// TIA Portal V20 export
FUNCTION "03 T4 LANT Aux" : Void   // FC1312, LAD
TITLE = AUXILIARIES
{ S7_Optimized_Access := 'TRUE' }
// stored: AutoNumber false, SetENOAutomatically false
   VAR_TEMP
      Aux_OS : Bool;
      Aux_sup : Real;
      Aux_inf : Real;
      Aux_DInt : DInt;
      Aux_Real : Real;
   END_VAR
   VAR CONSTANT
      "Max differenza L tubi" : Real := 500.0;
   END_VAR
   VAR_TEMP   // added for the SCL form of the ladder/FBD networks
      _w1 : Bool;
      _w2 : Bool;
   END_VAR
BEGIN

REGION Network 1: =========== MEMORIES ===========
END_REGION

REGION Network 2: TimeOutBancal: Calcul TimeOut
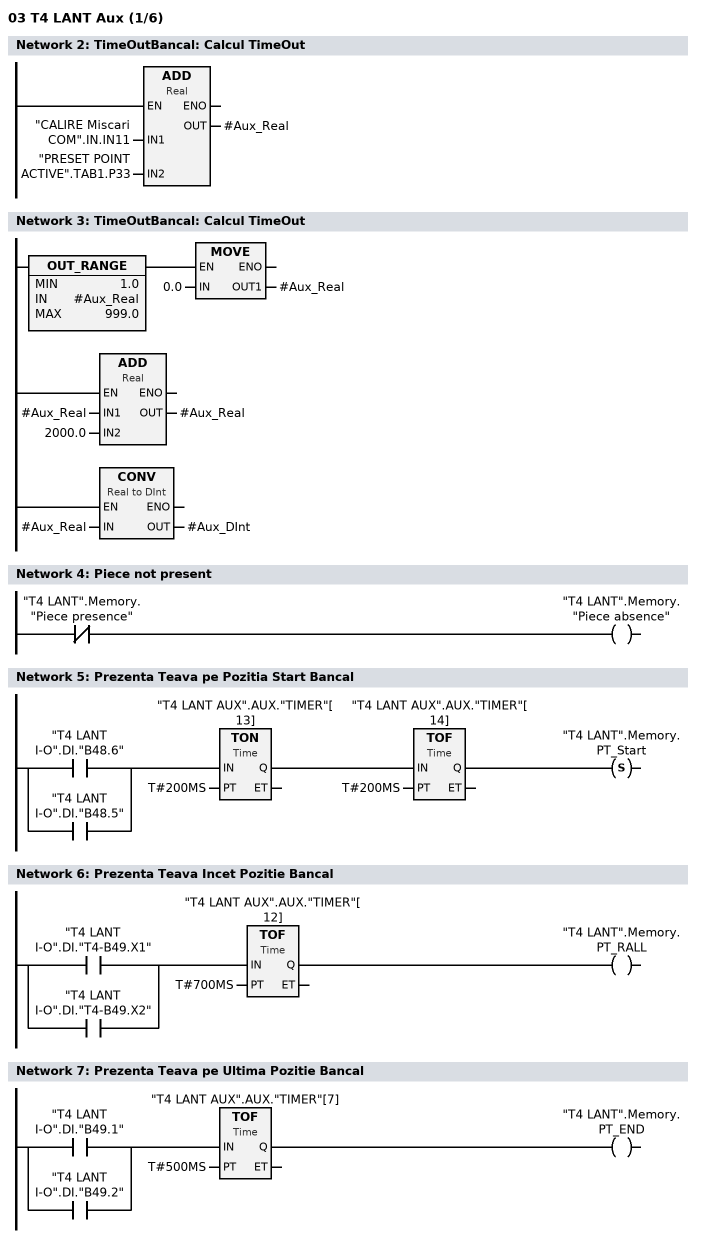
   RUNG wire#powerrail
      { S7_Templates := "SrcType := Real" } Add(in1 := "CALIRE Miscari COM".IN.IN11, in2 := "PRESET POINT ACTIVE".TAB1.P33, out => #Aux_Real)
   END_RUNG
   // the same network as SCL:
   #Aux_Real := "CALIRE Miscari COM".IN.IN11 + "PRESET POINT ACTIVE".TAB1.P33;
END_REGION

REGION Network 3: TimeOutBancal: Calcul TimeOut
   IF (#Aux_Real < 1.0) OR (#Aux_Real > 999.0) THEN #Aux_Real := 0.0; END_IF;
   #Aux_Real := #Aux_Real + 2000.0;
   #Aux_DInt := REAL_TO_DINT(#Aux_Real);
END_REGION

REGION Network 4: Piece not present
   RUNG wire#powerrail
      I_Contact( "T4 LANT".Memory."Piece presence" )
      Coil( "T4 LANT".Memory."Piece absence" )
   END_RUNG
   // the same network as SCL:
   "T4 LANT".Memory."Piece absence" := NOT "T4 LANT".Memory."Piece presence";
END_REGION

REGION Network 5: Prezenta Teava pe Pozitia Start Bancal
   RUNG wire#powerrail
      Contact( "T4 LANT I-O".DI."B48.6" )
      wire#w1
      { S7_Templates := "time_type := Time" } "T4 LANT AUX".AUX."TIMER"[13].TON(pt := T#200MS, et =>)
      { S7_Templates := "time_type := Time" } "T4 LANT AUX".AUX."TIMER"[14].TOF(pt := T#200MS, et =>)
      S_Coil( "T4 LANT".Memory.PT_Start )
   END_RUNG
   RUNG wire#powerrail
      Contact( "T4 LANT I-O".DI."B48.5" )
   END_RUNG wire#w1
   // the same network as SCL:
   "T4 LANT AUX".AUX."TIMER"[13].TON(IN := "T4 LANT I-O".DI."B48.6" OR "T4 LANT I-O".DI."B48.5", PT := T#200MS);
   "T4 LANT AUX".AUX."TIMER"[14].TOF(IN := "T4 LANT AUX".AUX."TIMER"[13].Q, PT := T#200MS);
   IF "T4 LANT AUX".AUX."TIMER"[14].Q THEN "T4 LANT".Memory.PT_Start := TRUE; END_IF;
END_REGION

REGION Network 6: Prezenta Teava Incet Pozitie Bancal
   RUNG wire#powerrail
      Contact( "T4 LANT I-O".DI."T4-B49.X1" )
      wire#w1
      { S7_Templates := "time_type := Time" } "T4 LANT AUX".AUX."TIMER"[12].TOF(pt := T#700MS, et =>)
      Coil( "T4 LANT".Memory.PT_RALL )
   END_RUNG
   RUNG wire#powerrail
      Contact( "T4 LANT I-O".DI."T4-B49.X2" )
   END_RUNG wire#w1
   // the same network as SCL:
   "T4 LANT AUX".AUX."TIMER"[12].TOF(IN := "T4 LANT I-O".DI."T4-B49.X1" OR "T4 LANT I-O".DI."T4-B49.X2",
                           PT := T#700MS);
   "T4 LANT".Memory.PT_RALL := "T4 LANT AUX".AUX."TIMER"[12].Q;
END_REGION

REGION Network 7: Prezenta Teava pe Ultima Pozitie Bancal
   RUNG wire#powerrail
      Contact( "T4 LANT I-O".DI."B49.1" )
      wire#w1
      { S7_Templates := "time_type := Time" } "T4 LANT AUX".AUX."TIMER"[7].TOF(pt := T#500MS, et =>)
      Coil( "T4 LANT".Memory.PT_END )
   END_RUNG
   RUNG wire#powerrail
      Contact( "T4 LANT I-O".DI."B49.2" )
   END_RUNG wire#w1
   // the same network as SCL:
   "T4 LANT AUX".AUX."TIMER"[7].TOF(IN := "T4 LANT I-O".DI."B49.1" OR "T4 LANT I-O".DI."B49.2", PT := T#500MS);
   "T4 LANT".Memory.PT_END := "T4 LANT AUX".AUX."TIMER"[7].Q;
END_REGION

REGION Network 8: T4-Lant: LAnt in Pozitia 'Pas'
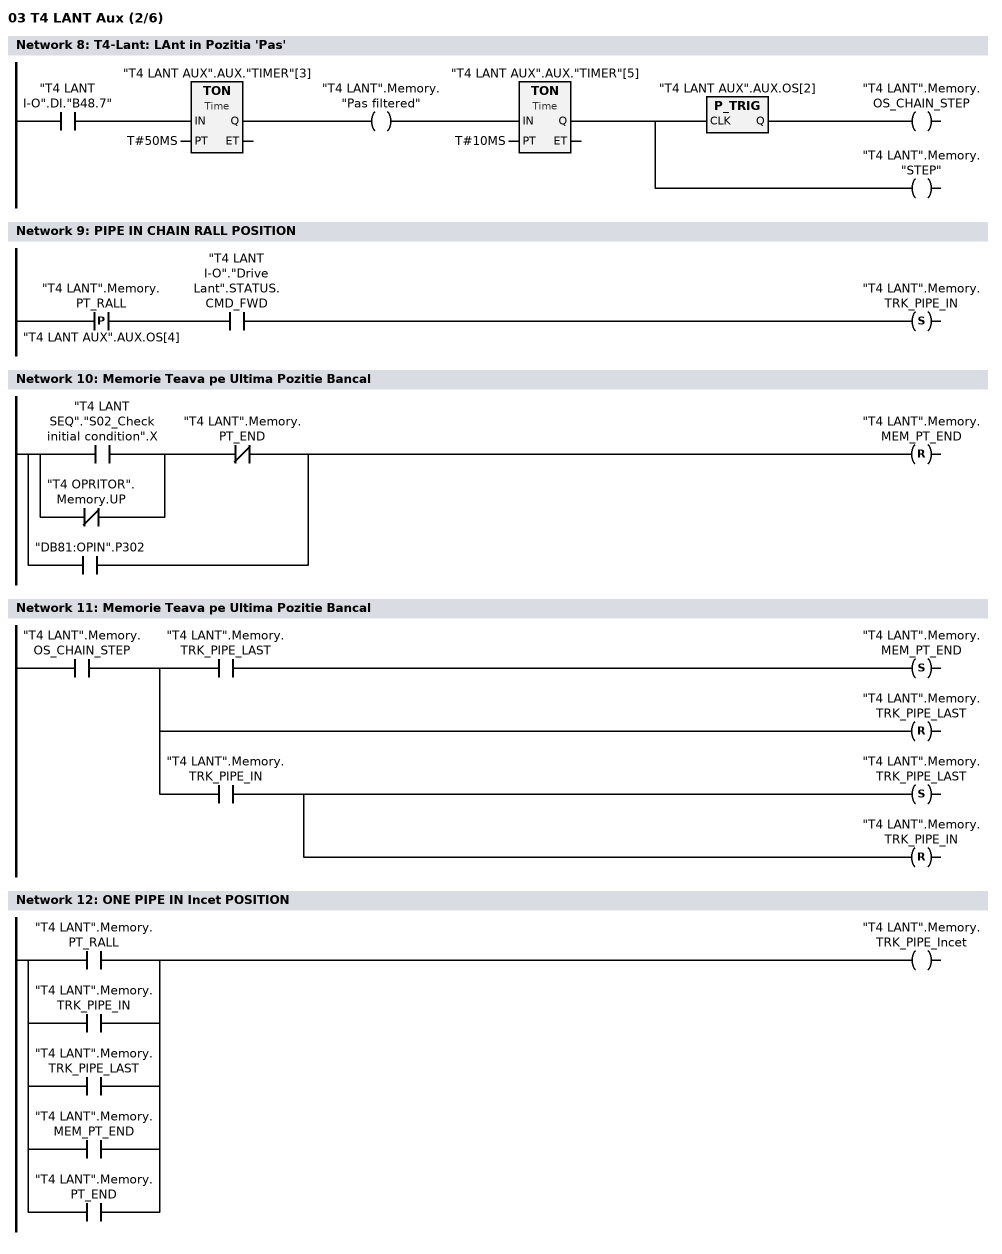
   RUNG wire#powerrail
      Contact( "T4 LANT I-O".DI."B48.7" )
      { S7_Templates := "time_type := Time" } "T4 LANT AUX".AUX."TIMER"[3].TON(pt := T#50MS, et =>)
      Coil( "T4 LANT".Memory."Pas filtered" )
      { S7_Templates := "time_type := Time" } "T4 LANT AUX".AUX."TIMER"[5].TON(pt := T#10MS, et =>)
      wire#w1
      P_Trig( "T4 LANT AUX".AUX.OS[2] )
      Coil( "T4 LANT".Memory.OS_CHAIN_STEP )
   END_RUNG
   RUNG wire#w1
      Coil( "T4 LANT".Memory."STEP" )
   END_RUNG
   // the same network as SCL:
   "T4 LANT AUX".AUX."TIMER"[3].TON(IN := "T4 LANT I-O".DI."B48.7", PT := T#50MS);
   "T4 LANT".Memory."Pas filtered" := "T4 LANT AUX".AUX."TIMER"[3].Q;
   "T4 LANT AUX".AUX."TIMER"[5].TON(IN := "T4 LANT AUX".AUX."TIMER"[3].Q, PT := T#10MS);
   #_w1 := "T4 LANT AUX".AUX."TIMER"[5].Q AND NOT "T4 LANT AUX".AUX.OS[2];   // rising edge
   "T4 LANT AUX".AUX.OS[2] := "T4 LANT AUX".AUX."TIMER"[5].Q;
   "T4 LANT".Memory.OS_CHAIN_STEP := #_w1;
   "T4 LANT".Memory."STEP" := "T4 LANT AUX".AUX."TIMER"[5].Q;
END_REGION

REGION Network 9: PIPE IN CHAIN RALL POSITION
   RUNG wire#powerrail
      P_Contact(operand := "T4 LANT".Memory.PT_RALL, bit := "T4 LANT AUX".AUX.OS[4])
      Contact( "T4 LANT I-O"."Drive Lant".STATUS.CMD_FWD )
      S_Coil( "T4 LANT".Memory.TRK_PIPE_IN )
   END_RUNG
   // the same network as SCL:
   #_w1 := "T4 LANT".Memory.PT_RALL AND NOT "T4 LANT AUX".AUX.OS[4];   // rising edge of "T4 LANT".Memory.PT_RALL
   "T4 LANT AUX".AUX.OS[4] := "T4 LANT".Memory.PT_RALL;
   IF #_w1 AND "T4 LANT I-O"."Drive Lant".STATUS.CMD_FWD THEN "T4 LANT".Memory.TRK_PIPE_IN := TRUE; END_IF;
END_REGION

REGION Network 10: Memorie Teava pe Ultima Pozitie Bancal
   RUNG wire#powerrail
      Contact( "T4 LANT SEQ"."S02_Check initial condition".X )
      wire#w1
      I_Contact( "T4 LANT".Memory.PT_END )
      wire#w2
      R_Coil( "T4 LANT".Memory.MEM_PT_END )
   END_RUNG
   RUNG wire#powerrail
      I_Contact( "T4 OPRITOR".Memory.UP )
   END_RUNG wire#w1
   RUNG wire#powerrail
      Contact( "DB81:OPIN".P302 )
   END_RUNG wire#w2
   // the same network as SCL:
   IF (("T4 LANT SEQ"."S02_Check initial condition".X OR NOT "T4 OPRITOR".Memory.UP) AND NOT "T4 LANT".Memory.PT_END) OR "DB81:OPIN".P302 THEN
       "T4 LANT".Memory.MEM_PT_END := FALSE;
   END_IF;
END_REGION

REGION Network 11: Memorie Teava pe Ultima Pozitie Bancal
   RUNG wire#powerrail
      Contact( "T4 LANT".Memory.OS_CHAIN_STEP )
      wire#w1
      Contact( "T4 LANT".Memory.TRK_PIPE_LAST )
      S_Coil( "T4 LANT".Memory.MEM_PT_END )
   END_RUNG
   RUNG wire#w1
      R_Coil( "T4 LANT".Memory.TRK_PIPE_LAST )
   END_RUNG
   RUNG wire#w1
      Contact( "T4 LANT".Memory.TRK_PIPE_IN )
      wire#w2
      S_Coil( "T4 LANT".Memory.TRK_PIPE_LAST )
   END_RUNG
   RUNG wire#w2
      R_Coil( "T4 LANT".Memory.TRK_PIPE_IN )
   END_RUNG
   // the same network as SCL:
   IF "T4 LANT".Memory.OS_CHAIN_STEP AND "T4 LANT".Memory.TRK_PIPE_LAST THEN
       "T4 LANT".Memory.MEM_PT_END := TRUE;
   END_IF;
   IF "T4 LANT".Memory.OS_CHAIN_STEP THEN "T4 LANT".Memory.TRK_PIPE_LAST := FALSE; END_IF;
   IF "T4 LANT".Memory.OS_CHAIN_STEP AND "T4 LANT".Memory.TRK_PIPE_IN THEN
       "T4 LANT".Memory.TRK_PIPE_LAST := TRUE;
       "T4 LANT".Memory.TRK_PIPE_IN := FALSE;
   END_IF;
END_REGION

REGION Network 12: ONE PIPE IN Incet POSITION
   RUNG wire#powerrail
      Contact( "T4 LANT".Memory.PT_RALL )
      wire#w1
      Coil( "T4 LANT".Memory.TRK_PIPE_Incet )
   END_RUNG
   RUNG wire#powerrail
      Contact( "T4 LANT".Memory.TRK_PIPE_IN )
   END_RUNG wire#w1
   RUNG wire#powerrail
      Contact( "T4 LANT".Memory.TRK_PIPE_LAST )
   END_RUNG wire#w1
   RUNG wire#powerrail
      Contact( "T4 LANT".Memory.MEM_PT_END )
   END_RUNG wire#w1
   RUNG wire#powerrail
      Contact( "T4 LANT".Memory.PT_END )
   END_RUNG wire#w1
   // the same network as SCL:
   "T4 LANT".Memory.TRK_PIPE_Incet := "T4 LANT".Memory.PT_RALL OR "T4 LANT".Memory.TRK_PIPE_IN OR "T4 LANT".Memory.TRK_PIPE_LAST OR "T4 LANT".Memory.MEM_PT_END OR "T4 LANT".Memory.PT_END;
END_REGION

REGION Network 13: 1 pipe to charge
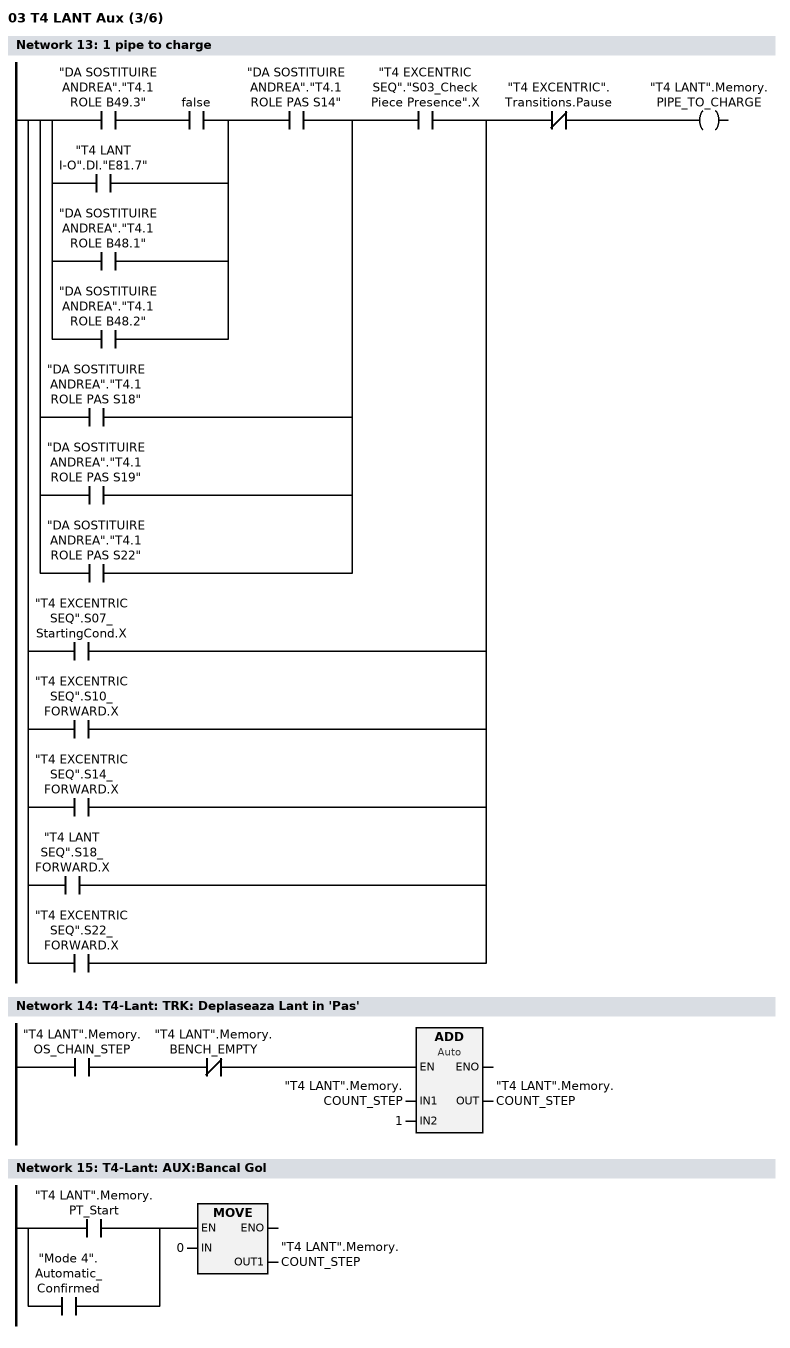
   RUNG wire#powerrail
      Contact( "DA SOSTITUIRE ANDREA"."T4.1 ROLE B49.3" )
      Contact( false )
      wire#w1
      Contact( "DA SOSTITUIRE ANDREA"."T4.1 ROLE PAS S14" )
      wire#w2
      Contact( "T4 EXCENTRIC SEQ"."S03_Check Piece Presence".X )
      wire#w3
      I_Contact( "T4 EXCENTRIC".Transitions.Pause )
      Coil( "T4 LANT".Memory.PIPE_TO_CHARGE )
   END_RUNG
   RUNG wire#powerrail
      Contact( "T4 LANT I-O".DI."E81.7" )
   END_RUNG wire#w1
   RUNG wire#powerrail
      Contact( "DA SOSTITUIRE ANDREA"."T4.1 ROLE B48.1" )
   END_RUNG wire#w1
   RUNG wire#powerrail
      Contact( "DA SOSTITUIRE ANDREA"."T4.1 ROLE B48.2" )
   END_RUNG wire#w1
   RUNG wire#powerrail
      Contact( "DA SOSTITUIRE ANDREA"."T4.1 ROLE PAS S18" )
   END_RUNG wire#w2
   RUNG wire#powerrail
      Contact( "DA SOSTITUIRE ANDREA"."T4.1 ROLE PAS S19" )
   END_RUNG wire#w2
   RUNG wire#powerrail
      Contact( "DA SOSTITUIRE ANDREA"."T4.1 ROLE PAS S22" )
   END_RUNG wire#w2
   RUNG wire#powerrail
      Contact( "T4 EXCENTRIC SEQ".S07_StartingCond.X )
   END_RUNG wire#w3
   RUNG wire#powerrail
      Contact( "T4 EXCENTRIC SEQ".S10_FORWARD.X )
   END_RUNG wire#w3
   RUNG wire#powerrail
      Contact( "T4 EXCENTRIC SEQ".S14_FORWARD.X )
   END_RUNG wire#w3
   RUNG wire#powerrail
      Contact( "T4 LANT SEQ".S18_FORWARD.X )
   END_RUNG wire#w3
   RUNG wire#powerrail
      Contact( "T4 EXCENTRIC SEQ".S22_FORWARD.X )
   END_RUNG wire#w3
   // the same network as SCL:
   "T4 LANT".Memory.PIPE_TO_CHARGE := (((((("DA SOSTITUIRE ANDREA"."T4.1 ROLE B49.3" AND false) OR "T4 LANT I-O".DI."E81.7" OR "DA SOSTITUIRE ANDREA"."T4.1 ROLE B48.1" OR "DA SOSTITUIRE ANDREA"."T4.1 ROLE B48.2") AND "DA SOSTITUIRE ANDREA"."T4.1 ROLE PAS S14") OR "DA SOSTITUIRE ANDREA"."T4.1 ROLE PAS S18" OR "DA SOSTITUIRE ANDREA"."T4.1 ROLE PAS S19" OR "DA SOSTITUIRE ANDREA"."T4.1 ROLE PAS S22") AND "T4 EXCENTRIC SEQ"."S03_Check Piece Presence".X) OR "T4 EXCENTRIC SEQ".S07_StartingCond.X OR "T4 EXCENTRIC SEQ".S10_FORWARD.X OR "T4 EXCENTRIC SEQ".S14_FORWARD.X OR "T4 LANT SEQ".S18_FORWARD.X OR "T4 EXCENTRIC SEQ".S22_FORWARD.X) AND NOT "T4 EXCENTRIC".Transitions.Pause;
END_REGION

REGION Network 14: T4-Lant: TRK: Deplaseaza Lant in 'Pas'
   RUNG wire#powerrail
      Contact( "T4 LANT".Memory.OS_CHAIN_STEP )
      I_Contact( "T4 LANT".Memory.BENCH_EMPTY )
      Add(in1 := "T4 LANT".Memory.COUNT_STEP, in2 := 1, out => "T4 LANT".Memory.COUNT_STEP)
   END_RUNG
   // the same network as SCL:
   IF "T4 LANT".Memory.OS_CHAIN_STEP AND NOT "T4 LANT".Memory.BENCH_EMPTY THEN
       "T4 LANT".Memory.COUNT_STEP := "T4 LANT".Memory.COUNT_STEP + 1;
   END_IF;
END_REGION

REGION Network 15: T4-Lant: AUX:Bancal Gol
   RUNG wire#powerrail
      Contact( "T4 LANT".Memory.PT_Start )
      wire#w1
      Move(in := 0, out1 => "T4 LANT".Memory.COUNT_STEP)
   END_RUNG
   RUNG wire#powerrail
      Contact( "Mode 4".Automatic_Confirmed )
   END_RUNG wire#w1
   // the same network as SCL:
   IF "T4 LANT".Memory.PT_Start OR "Mode 4".Automatic_Confirmed THEN
       "T4 LANT".Memory.COUNT_STEP := 0;
   END_IF;
END_REGION

REGION Network 16: T4-Lant: AUX:Bancal Gol
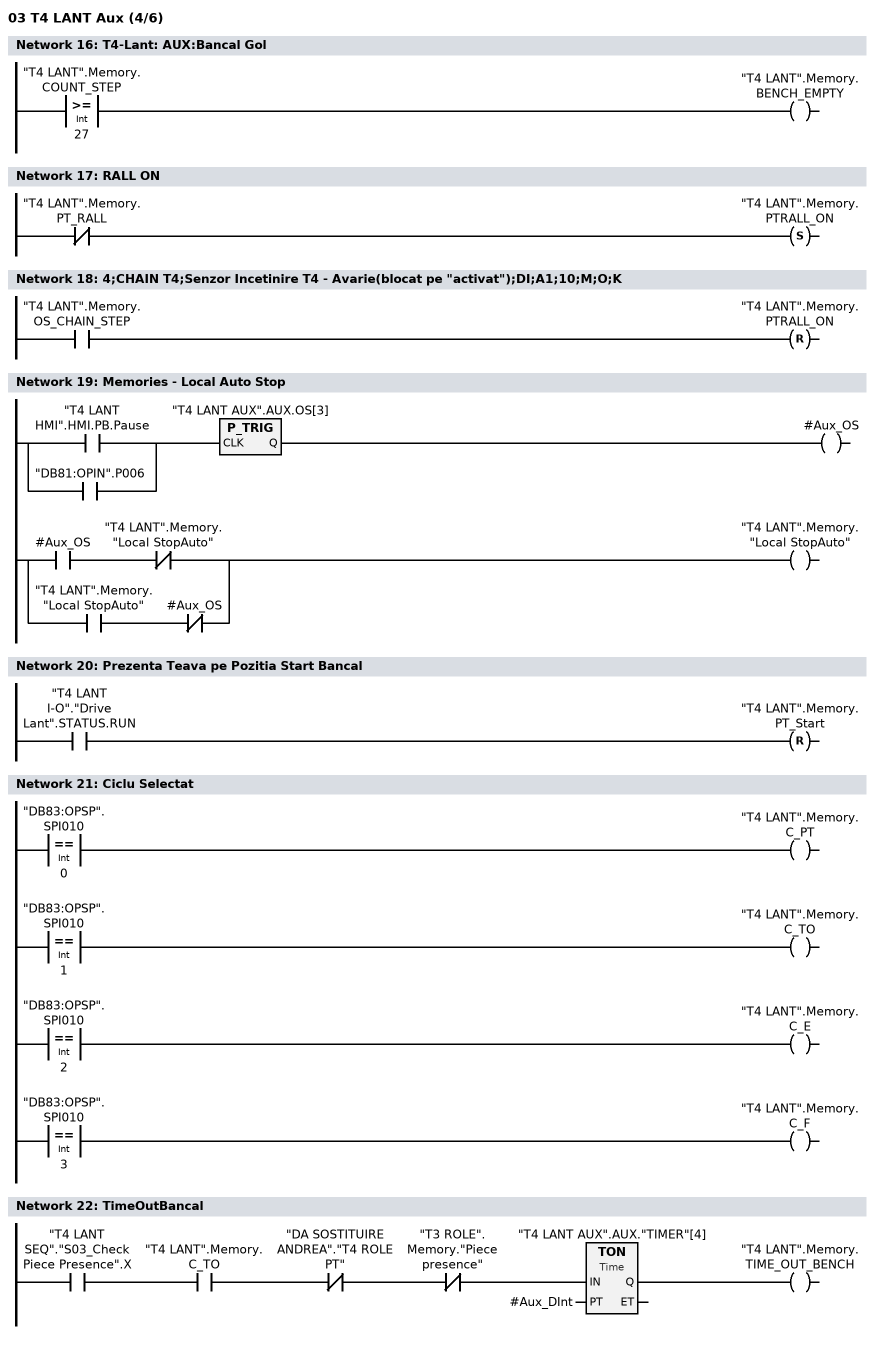
   RUNG wire#powerrail
      { S7_Templates := "SrcType := Int" } GE_Contact(in1 := "T4 LANT".Memory.COUNT_STEP, in2 := 27)
      Coil( "T4 LANT".Memory.BENCH_EMPTY )
   END_RUNG
   // the same network as SCL:
   "T4 LANT".Memory.BENCH_EMPTY := "T4 LANT".Memory.COUNT_STEP >= 27;
END_REGION

REGION Network 17: RALL ON
   RUNG wire#powerrail
      I_Contact( "T4 LANT".Memory.PT_RALL )
      S_Coil( "T4 LANT".Memory.PTRALL_ON )
   END_RUNG
   // the same network as SCL:
   IF NOT "T4 LANT".Memory.PT_RALL THEN "T4 LANT".Memory.PTRALL_ON := TRUE; END_IF;
END_REGION

REGION Network 18: 4;CHAIN T4;Senzor Incetinire T4 - Avarie(blocat pe "activat");DI;A1;10;M;O;K
   RUNG wire#powerrail
      Contact( "T4 LANT".Memory.OS_CHAIN_STEP )
      R_Coil( "T4 LANT".Memory.PTRALL_ON )
   END_RUNG
   // the same network as SCL:
   IF "T4 LANT".Memory.OS_CHAIN_STEP THEN "T4 LANT".Memory.PTRALL_ON := FALSE; END_IF;
END_REGION

REGION Network 19: Memories - Local Auto Stop
   RUNG wire#powerrail
      Contact( "T4 LANT HMI".HMI.PB.Pause )
      wire#w1
      P_Trig( "T4 LANT AUX".AUX.OS[3] )
      Coil( #Aux_OS )
   END_RUNG
   RUNG wire#powerrail
      Contact( "DB81:OPIN".P006 )
   END_RUNG wire#w1
   RUNG wire#powerrail
      Contact( #Aux_OS )
      I_Contact( "T4 LANT".Memory."Local StopAuto" )
      wire#w2
      Coil( "T4 LANT".Memory."Local StopAuto" )
   END_RUNG
   RUNG wire#powerrail
      Contact( "T4 LANT".Memory."Local StopAuto" )
      I_Contact( #Aux_OS )
   END_RUNG wire#w2
   // the same network as SCL:
   #_w1 := "T4 LANT HMI".HMI.PB.Pause OR "DB81:OPIN".P006;
   #_w2 := #_w1 AND NOT "T4 LANT AUX".AUX.OS[3];   // rising edge
   "T4 LANT AUX".AUX.OS[3] := #_w1;
   #Aux_OS := #_w2;
   "T4 LANT".Memory."Local StopAuto" := (#Aux_OS AND NOT "T4 LANT".Memory."Local StopAuto") OR ("T4 LANT".Memory."Local StopAuto" AND NOT #Aux_OS);
END_REGION

REGION Network 20: Prezenta Teava pe Pozitia Start Bancal
   RUNG wire#powerrail
      Contact( "T4 LANT I-O"."Drive Lant".STATUS.RUN )
      R_Coil( "T4 LANT".Memory.PT_Start )
   END_RUNG
   // the same network as SCL:
   IF "T4 LANT I-O"."Drive Lant".STATUS.RUN THEN "T4 LANT".Memory.PT_Start := FALSE; END_IF;
END_REGION

REGION Network 21: Ciclu Selectat
   RUNG wire#powerrail
      { S7_Templates := "SrcType := Int" } EQ_Contact(in1 := "DB83:OPSP".SPI010, in2 := 0)
      Coil( "T4 LANT".Memory.C_PT )
   END_RUNG
   RUNG wire#powerrail
      { S7_Templates := "SrcType := Int" } EQ_Contact(in1 := "DB83:OPSP".SPI010, in2 := 1)
      Coil( "T4 LANT".Memory.C_TO )
   END_RUNG
   RUNG wire#powerrail
      { S7_Templates := "SrcType := Int" } EQ_Contact(in1 := "DB83:OPSP".SPI010, in2 := 2)
      Coil( "T4 LANT".Memory.C_E )
   END_RUNG
   RUNG wire#powerrail
      { S7_Templates := "SrcType := Int" } EQ_Contact(in1 := "DB83:OPSP".SPI010, in2 := 3)
      Coil( "T4 LANT".Memory.C_F )
   END_RUNG
   // the same network as SCL:
   "T4 LANT".Memory.C_PT := "DB83:OPSP".SPI010 = 0;
   "T4 LANT".Memory.C_TO := "DB83:OPSP".SPI010 = 1;
   "T4 LANT".Memory.C_E := "DB83:OPSP".SPI010 = 2;
   "T4 LANT".Memory.C_F := "DB83:OPSP".SPI010 = 3;
END_REGION

REGION Network 22: TimeOutBancal
   RUNG wire#powerrail
      Contact( "T4 LANT SEQ"."S03_Check Piece Presence".X )
      Contact( "T4 LANT".Memory.C_TO )
      I_Contact( "DA SOSTITUIRE ANDREA"."T4 ROLE PT" )
      I_Contact( "T3 ROLE".Memory."Piece presence" )
      { S7_Templates := "time_type := Time" } "T4 LANT AUX".AUX."TIMER"[4].TON(pt := #Aux_DInt, et =>)
      Coil( "T4 LANT".Memory.TIME_OUT_BENCH )
   END_RUNG
   // the same network as SCL:
   "T4 LANT AUX".AUX."TIMER"[4].TON(IN := "T4 LANT SEQ"."S03_Check Piece Presence".X AND "T4 LANT".Memory.C_TO AND NOT "DA SOSTITUIRE ANDREA"."T4 ROLE PT" AND NOT "T3 ROLE".Memory."Piece presence",
                           PT := #Aux_DInt);
   "T4 LANT".Memory.TIME_OUT_BENCH := "T4 LANT AUX".AUX."TIMER"[4].Q;
END_REGION

REGION Network 23: Lant T4 Pasi
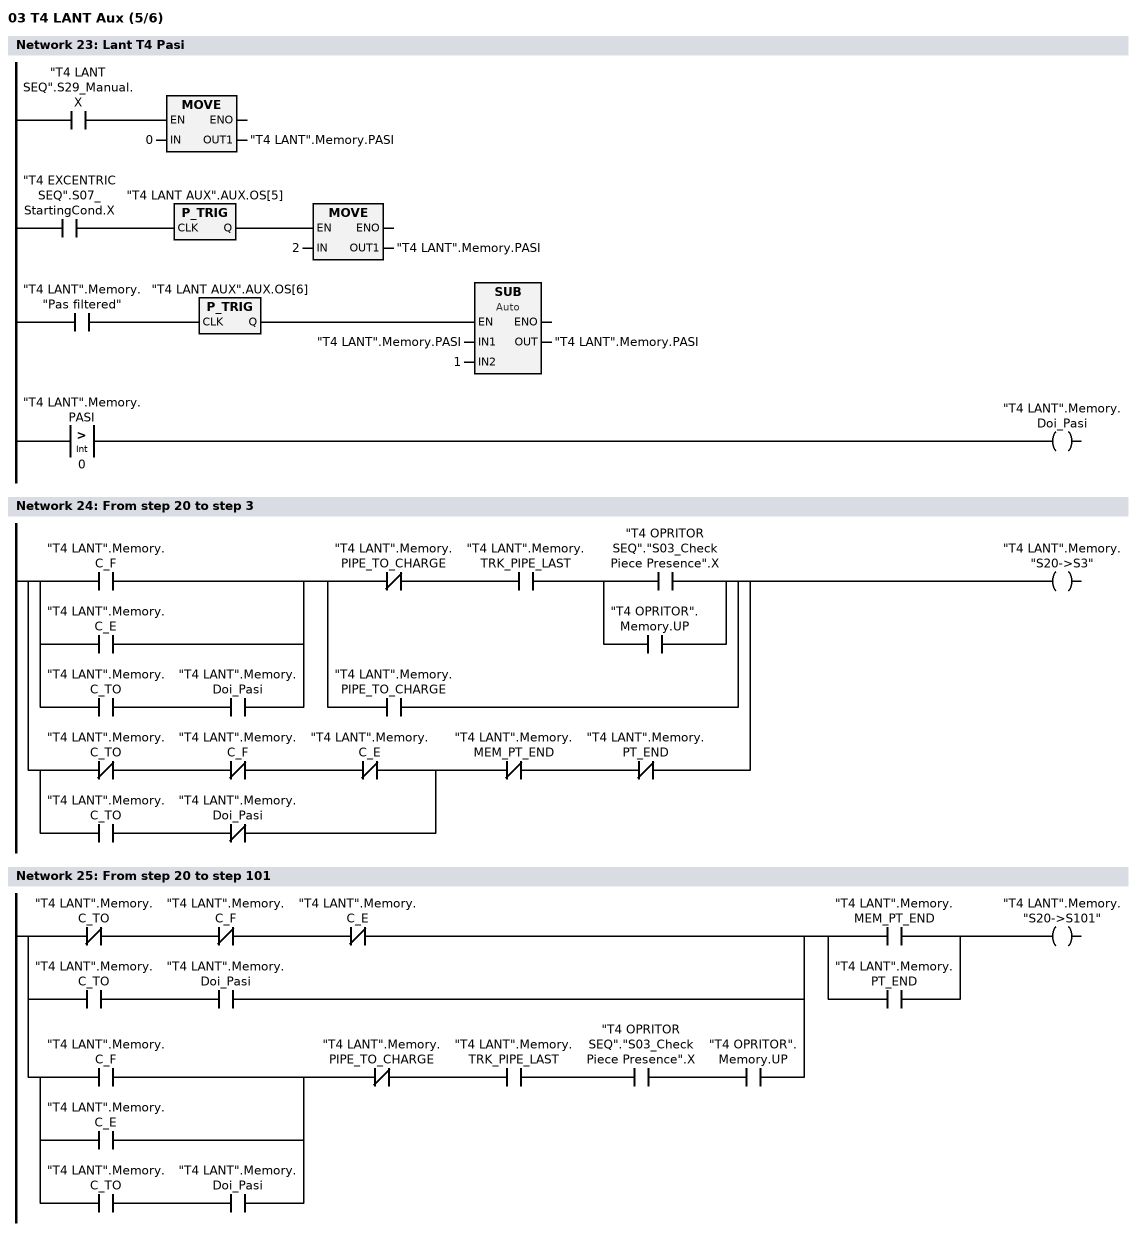
   RUNG wire#powerrail
      Contact( "T4 LANT SEQ".S29_Manual.X )
      Move(in := 0, out1 => "T4 LANT".Memory.PASI)
   END_RUNG
   RUNG wire#powerrail
      Contact( "T4 EXCENTRIC SEQ".S07_StartingCond.X )
      P_Trig( "T4 LANT AUX".AUX.OS[5] )
      Move(in := 2, out1 => "T4 LANT".Memory.PASI)
   END_RUNG
   RUNG wire#powerrail
      Contact( "T4 LANT".Memory."Pas filtered" )
      P_Trig( "T4 LANT AUX".AUX.OS[6] )
      Sub(in1 := "T4 LANT".Memory.PASI, in2 := 1, out => "T4 LANT".Memory.PASI)
   END_RUNG
   RUNG wire#powerrail
      { S7_Templates := "SrcType := Int" } GT_Contact(in1 := "T4 LANT".Memory.PASI, in2 := 0)
      Coil( "T4 LANT".Memory.Doi_Pasi )
   END_RUNG
   // the same network as SCL:
   IF "T4 LANT SEQ".S29_Manual.X THEN "T4 LANT".Memory.PASI := 0; END_IF;
   #_w1 := "T4 EXCENTRIC SEQ".S07_StartingCond.X AND NOT "T4 LANT AUX".AUX.OS[5];   // rising edge
   "T4 LANT AUX".AUX.OS[5] := "T4 EXCENTRIC SEQ".S07_StartingCond.X;
   IF #_w1 THEN "T4 LANT".Memory.PASI := 2; END_IF;
   #_w2 := "T4 LANT".Memory."Pas filtered" AND NOT "T4 LANT AUX".AUX.OS[6];   // rising edge
   "T4 LANT AUX".AUX.OS[6] := "T4 LANT".Memory."Pas filtered";
   IF #_w2 THEN "T4 LANT".Memory.PASI := "T4 LANT".Memory.PASI - 1; END_IF;
   "T4 LANT".Memory.Doi_Pasi := "T4 LANT".Memory.PASI > 0;
END_REGION

REGION Network 24: From step 20 to step 3
   RUNG wire#powerrail
      Contact( "T4 LANT".Memory.C_F )
      wire#w1
      I_Contact( "T4 LANT".Memory.PIPE_TO_CHARGE )
      Contact( "T4 LANT".Memory.TRK_PIPE_LAST )
      wire#w2
      Contact( "T4 OPRITOR SEQ"."S03_Check Piece Presence".X )
      wire#w3
      Coil( "T4 LANT".Memory."S20->S3" )
   END_RUNG
   RUNG wire#powerrail
      Contact( "T4 LANT".Memory.C_E )
   END_RUNG wire#w1
   RUNG wire#powerrail
      Contact( "T4 LANT".Memory.C_TO )
      Contact( "T4 LANT".Memory.Doi_Pasi )
   END_RUNG wire#w1
   RUNG wire#w2
      Contact( "T4 OPRITOR".Memory.UP )
   END_RUNG wire#w3
   RUNG wire#w1
      Contact( "T4 LANT".Memory.PIPE_TO_CHARGE )
   END_RUNG wire#w3
   RUNG wire#powerrail
      I_Contact( "T4 LANT".Memory.C_TO )
      I_Contact( "T4 LANT".Memory.C_F )
      I_Contact( "T4 LANT".Memory.C_E )
      wire#w4
      I_Contact( "T4 LANT".Memory.MEM_PT_END )
      I_Contact( "T4 LANT".Memory.PT_END )
   END_RUNG wire#w3
   RUNG wire#powerrail
      Contact( "T4 LANT".Memory.C_TO )
      I_Contact( "T4 LANT".Memory.Doi_Pasi )
   END_RUNG wire#w4
   // the same network as SCL:
   "T4 LANT".Memory."S20->S3" := (("T4 LANT".Memory.C_F OR "T4 LANT".Memory.C_E OR ("T4 LANT".Memory.C_TO AND "T4 LANT".Memory.Doi_Pasi)) AND ((NOT "T4 LANT".Memory.PIPE_TO_CHARGE AND "T4 LANT".Memory.TRK_PIPE_LAST AND ("T4 OPRITOR SEQ"."S03_Check Piece Presence".X OR "T4 OPRITOR".Memory.UP)) OR "T4 LANT".Memory.PIPE_TO_CHARGE)) OR (((NOT "T4 LANT".Memory.C_TO AND NOT "T4 LANT".Memory.C_F AND NOT "T4 LANT".Memory.C_E) OR ("T4 LANT".Memory.C_TO AND NOT "T4 LANT".Memory.Doi_Pasi)) AND NOT "T4 LANT".Memory.MEM_PT_END AND NOT "T4 LANT".Memory.PT_END);
END_REGION

REGION Network 25: From step 20 to step 101
   RUNG wire#powerrail
      I_Contact( "T4 LANT".Memory.C_TO )
      I_Contact( "T4 LANT".Memory.C_F )
      I_Contact( "T4 LANT".Memory.C_E )
      wire#w1
      Contact( "T4 LANT".Memory.MEM_PT_END )
      wire#w3
      Coil( "T4 LANT".Memory."S20->S101" )
   END_RUNG
   RUNG wire#powerrail
      Contact( "T4 LANT".Memory.C_TO )
      Contact( "T4 LANT".Memory.Doi_Pasi )
   END_RUNG wire#w1
   RUNG wire#powerrail
      Contact( "T4 LANT".Memory.C_F )
      wire#w2
      I_Contact( "T4 LANT".Memory.PIPE_TO_CHARGE )
      Contact( "T4 LANT".Memory.TRK_PIPE_LAST )
      Contact( "T4 OPRITOR SEQ"."S03_Check Piece Presence".X )
      Contact( "T4 OPRITOR".Memory.UP )
   END_RUNG wire#w1
   RUNG wire#powerrail
      Contact( "T4 LANT".Memory.C_E )
   END_RUNG wire#w2
   RUNG wire#powerrail
      Contact( "T4 LANT".Memory.C_TO )
      Contact( "T4 LANT".Memory.Doi_Pasi )
   END_RUNG wire#w2
   RUNG wire#w1
      Contact( "T4 LANT".Memory.PT_END )
   END_RUNG wire#w3
   // the same network as SCL:
   "T4 LANT".Memory."S20->S101" := ((NOT "T4 LANT".Memory.C_TO AND NOT "T4 LANT".Memory.C_F AND NOT "T4 LANT".Memory.C_E) OR ("T4 LANT".Memory.C_TO AND "T4 LANT".Memory.Doi_Pasi) OR (("T4 LANT".Memory.C_F OR "T4 LANT".Memory.C_E OR ("T4 LANT".Memory.C_TO AND "T4 LANT".Memory.Doi_Pasi)) AND NOT "T4 LANT".Memory.PIPE_TO_CHARGE AND "T4 LANT".Memory.TRK_PIPE_LAST AND "T4 OPRITOR SEQ"."S03_Check Piece Presence".X AND "T4 OPRITOR".Memory.UP)) AND ("T4 LANT".Memory.MEM_PT_END OR "T4 LANT".Memory.PT_END);
END_REGION

REGION Network 26: From step 20 to step 10
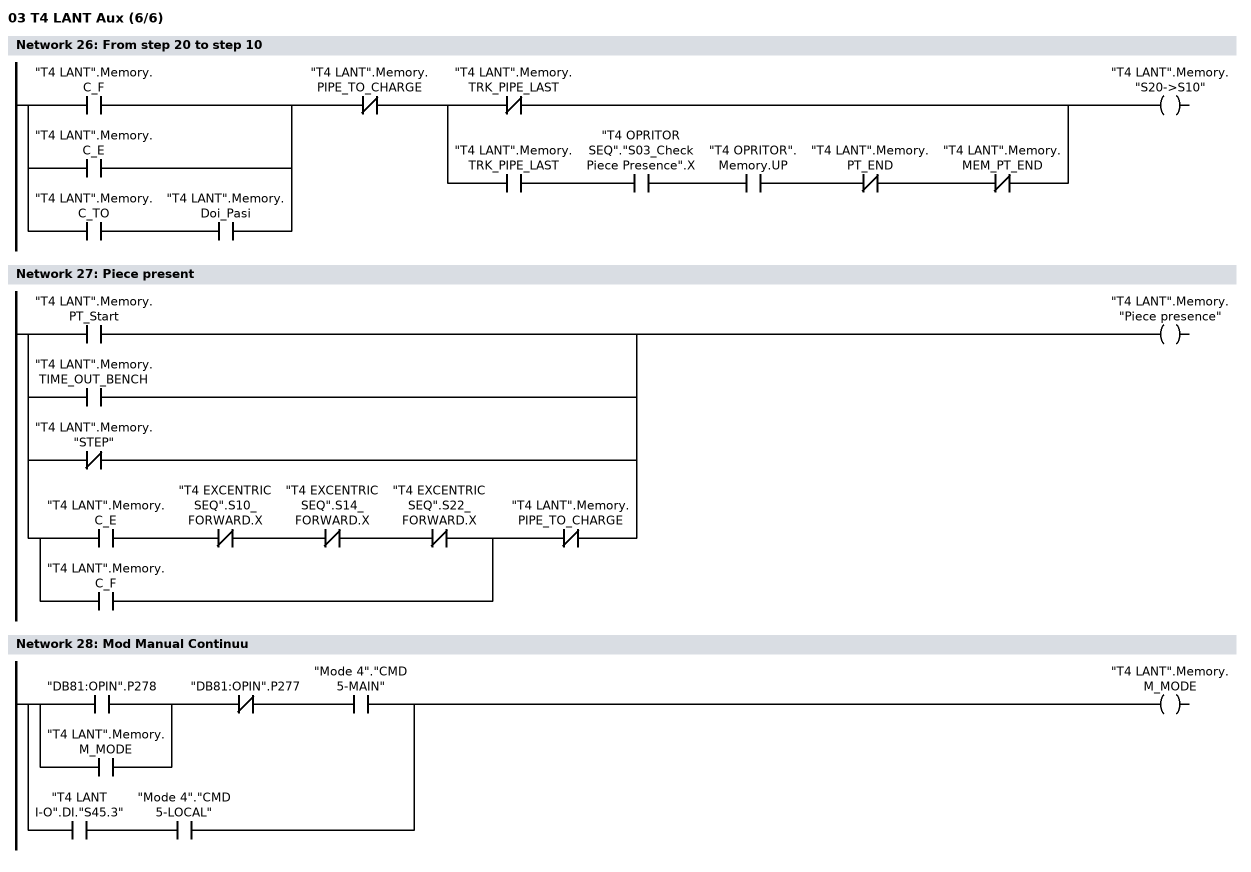
   RUNG wire#powerrail
      Contact( "T4 LANT".Memory.C_F )
      wire#w1
      I_Contact( "T4 LANT".Memory.PIPE_TO_CHARGE )
      wire#w2
      I_Contact( "T4 LANT".Memory.TRK_PIPE_LAST )
      wire#w3
      Coil( "T4 LANT".Memory."S20->S10" )
   END_RUNG
   RUNG wire#powerrail
      Contact( "T4 LANT".Memory.C_E )
   END_RUNG wire#w1
   RUNG wire#powerrail
      Contact( "T4 LANT".Memory.C_TO )
      Contact( "T4 LANT".Memory.Doi_Pasi )
   END_RUNG wire#w1
   RUNG wire#w2
      Contact( "T4 LANT".Memory.TRK_PIPE_LAST )
      Contact( "T4 OPRITOR SEQ"."S03_Check Piece Presence".X )
      Contact( "T4 OPRITOR".Memory.UP )
      I_Contact( "T4 LANT".Memory.PT_END )
      I_Contact( "T4 LANT".Memory.MEM_PT_END )
   END_RUNG wire#w3
   // the same network as SCL:
   "T4 LANT".Memory."S20->S10" := ("T4 LANT".Memory.C_F OR "T4 LANT".Memory.C_E OR ("T4 LANT".Memory.C_TO AND "T4 LANT".Memory.Doi_Pasi)) AND NOT "T4 LANT".Memory.PIPE_TO_CHARGE AND (NOT "T4 LANT".Memory.TRK_PIPE_LAST OR ("T4 LANT".Memory.TRK_PIPE_LAST AND "T4 OPRITOR SEQ"."S03_Check Piece Presence".X AND "T4 OPRITOR".Memory.UP AND NOT "T4 LANT".Memory.PT_END AND NOT "T4 LANT".Memory.MEM_PT_END));
END_REGION

REGION Network 27: Piece present
   RUNG wire#powerrail
      Contact( "T4 LANT".Memory.PT_Start )
      wire#w1
      Coil( "T4 LANT".Memory."Piece presence" )
   END_RUNG
   RUNG wire#powerrail
      Contact( "T4 LANT".Memory.TIME_OUT_BENCH )
   END_RUNG wire#w1
   RUNG wire#powerrail
      I_Contact( "T4 LANT".Memory."STEP" )
   END_RUNG wire#w1
   RUNG wire#powerrail
      Contact( "T4 LANT".Memory.C_E )
      I_Contact( "T4 EXCENTRIC SEQ".S10_FORWARD.X )
      I_Contact( "T4 EXCENTRIC SEQ".S14_FORWARD.X )
      I_Contact( "T4 EXCENTRIC SEQ".S22_FORWARD.X )
      wire#w2
      I_Contact( "T4 LANT".Memory.PIPE_TO_CHARGE )
   END_RUNG wire#w1
   RUNG wire#powerrail
      Contact( "T4 LANT".Memory.C_F )
   END_RUNG wire#w2
   // the same network as SCL:
   "T4 LANT".Memory."Piece presence" := "T4 LANT".Memory.PT_Start OR "T4 LANT".Memory.TIME_OUT_BENCH OR NOT "T4 LANT".Memory."STEP" OR ((("T4 LANT".Memory.C_E AND NOT "T4 EXCENTRIC SEQ".S10_FORWARD.X AND NOT "T4 EXCENTRIC SEQ".S14_FORWARD.X AND NOT "T4 EXCENTRIC SEQ".S22_FORWARD.X) OR "T4 LANT".Memory.C_F) AND NOT "T4 LANT".Memory.PIPE_TO_CHARGE);
END_REGION

REGION Network 28: Mod Manual Continuu
   RUNG wire#powerrail
      Contact( "DB81:OPIN".P278 )
      wire#w1
      I_Contact( "DB81:OPIN".P277 )
      Contact( "Mode 4"."CMD 5-MAIN" )
      wire#w2
      Coil( "T4 LANT".Memory.M_MODE )
   END_RUNG
   RUNG wire#powerrail
      Contact( "T4 LANT".Memory.M_MODE )
   END_RUNG wire#w1
   RUNG wire#powerrail
      Contact( "T4 LANT I-O".DI."S45.3" )
      Contact( "Mode 4"."CMD 5-LOCAL" )
   END_RUNG wire#w2
   // the same network as SCL:
   "T4 LANT".Memory.M_MODE := (("DB81:OPIN".P278 OR "T4 LANT".Memory.M_MODE) AND NOT "DB81:OPIN".P277 AND "Mode 4"."CMD 5-MAIN") OR ("T4 LANT I-O".DI."S45.3" AND "Mode 4"."CMD 5-LOCAL");
END_REGION
END_FUNCTION
